// TIA Portal V20 export
FUNCTION_BLOCK "Simulation"   // FB102, LAD
// stored: MemoryReserve 100, Namespace Unit1.Em3, SetENOAutomatically false
   VAR
      Simulation_addon_Instance { S7_SetPoint := 'True'} : "Simulation_addon";
   END_VAR
BEGIN

REGION Network 1: cmDancerEncoderAnalogInput
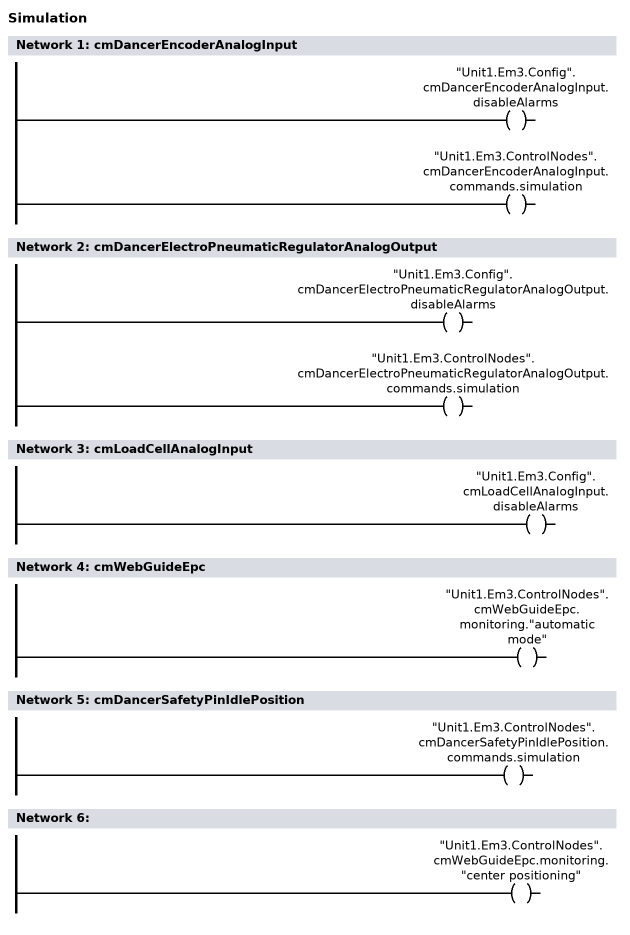
   RUNG wire#powerrail
      Coil( "Unit1.Em3.Config".cmDancerEncoderAnalogInput.disableAlarms )
   END_RUNG
   RUNG wire#powerrail
      Coil( "Unit1.Em3.ControlNodes".cmDancerEncoderAnalogInput.commands.simulation )
   END_RUNG
   // the same network as SCL:
   "Unit1.Em3.Config".cmDancerEncoderAnalogInput.disableAlarms := TRUE;
   "Unit1.Em3.ControlNodes".cmDancerEncoderAnalogInput.commands.simulation := TRUE;
END_REGION

REGION Network 2: cmDancerElectroPneumaticRegulatorAnalogOutput
   RUNG wire#powerrail
      Coil( "Unit1.Em3.Config".cmDancerElectroPneumaticRegulatorAnalogOutput.disableAlarms )
   END_RUNG
   RUNG wire#powerrail
      Coil( "Unit1.Em3.ControlNodes".cmDancerElectroPneumaticRegulatorAnalogOutput.commands.simulation )
   END_RUNG
   // the same network as SCL:
   "Unit1.Em3.Config".cmDancerElectroPneumaticRegulatorAnalogOutput.disableAlarms := TRUE;
   "Unit1.Em3.ControlNodes".cmDancerElectroPneumaticRegulatorAnalogOutput.commands.simulation := TRUE;
END_REGION

REGION Network 3: cmLoadCellAnalogInput
   RUNG wire#powerrail
      Coil( "Unit1.Em3.Config".cmLoadCellAnalogInput.disableAlarms )
   END_RUNG
   // the same network as SCL:
   "Unit1.Em3.Config".cmLoadCellAnalogInput.disableAlarms := TRUE;
END_REGION

REGION Network 4: cmWebGuideEpc
   RUNG wire#powerrail
      Coil( "Unit1.Em3.ControlNodes".cmWebGuideEpc.monitoring."automatic mode" )
   END_RUNG
   // the same network as SCL:
   "Unit1.Em3.ControlNodes".cmWebGuideEpc.monitoring."automatic mode" := TRUE;
END_REGION

REGION Network 5: cmDancerSafetyPinIdlePosition
   RUNG wire#powerrail
      Coil( "Unit1.Em3.ControlNodes".cmDancerSafetyPinIdlePosition.commands.simulation )
   END_RUNG
   // the same network as SCL:
   "Unit1.Em3.ControlNodes".cmDancerSafetyPinIdlePosition.commands.simulation := TRUE;
END_REGION

REGION Network 6
   RUNG wire#powerrail
      Coil( "Unit1.Em3.ControlNodes".cmWebGuideEpc.monitoring."center positioning" )
   END_RUNG
   // the same network as SCL:
   "Unit1.Em3.ControlNodes".cmWebGuideEpc.monitoring."center positioning" := TRUE;
END_REGION
END_FUNCTION_BLOCK
